FUNCTION_BLOCK MC_MoveAbsolute
VAR_INPUT
	Axis: AXIS_REF;
	
END_VAR
VAR_OUTPUT
END_VAR
VAR
END_VAR

Axis.ReadStatus();

END_FUNCTION_BLOCK

(* stored: Version 1.1.0.1, ProductVersion 3.1.4022.12
   POU MC_MoveAbsolute: Id {95b183ec-aab7-41f3-b788-80cdea153fa6}, SpecialFunc None *)
